# EPICS alarm handler configuration: alh_files/mgnt_li28.alhConfig
GROUP NULL MGNT:LI28:1
   $COMMAND edm -x -eolc -noedit mgnt_li28_main.edl

$ALIAS LI28
$GUIDANCE
LI28 Magnets
   Group Name: MGNT:LI28:1
   Summary PV:  MGNT:LI28:1:STATSUMY
$END

   INCLUDE MGNT:LI28:1 ./mgnt_li28_lgps.alhConfig
   INCLUDE MGNT:LI28:1 ./mgnt_li28_quad.alhConfig
   INCLUDE MGNT:LI28:1 ./mgnt_li28_xcor.alhConfig
   INCLUDE MGNT:LI28:1 ./mgnt_li28_ycor.alhConfig
